// TIA Portal V16 export
// export: Created 2022-11-14T17:35:46.2709233Z, ExportSetting WithDefaults, DisplayName Totally Integrated Automation Portal, DisplayVersion V16, DisplayName TIA Portal Version Control Interface, DisplayVersion V16, DisplayName TIA Portal Openness, DisplayVersion V16, DisplayName STEP 7 Professional, DisplayVersion V16, DisplayName STEP 7 Safety, DisplayVersion V16, DisplayName WinCC Advanced, DisplayVersion V16
DATA_BLOCK "DB234_Program16"   // DB234
{ S7_Optimized_Access := 'FALSE' }
AUTHOR : Robopac
VERSION : 0.0
// stored: AutoNumber false, IsOnlyStoredInLoadMemory false, IsWriteProtectedInAS false
   VAR RETAIN
      Program16 { S7_SetPoint := 'True'} : "DatiProgramma";
   END_VAR
BEGIN
   Program16.Wrapping := FALSE;
   Program16.TopLenght := 0;
   Program16.TopRelease := 0;
   Program16.TopDown := 0;
   Program16.Top := 0;
   Program16.PressurePTime := 0;
   Program16.LifterTime := 0;
   Program16.RevOverContrast := 0;
   Program16.RopeEndCycle := 16#00;
   Program16.Spare4 := 16#00;
   Program16.RopeTime := 0;
   Program16.RevOverClamp := 0;
   Program16.FilmForceFinalRev := 0;
   Program16.FilmPrestretchFinalRev := 0;
   Program16.ArmSpeed := 0;
   Program16.CarriageDown4Top := 0;
   Program16.TopDownTime := 0;
   Program16.LapsUnderTop := 0;
   Program16.Spare6 := 0;
   Program16.Spare7 := 0;
   Program16.Spare8 := 0;
   Program16.Spare9 := 0;
   Program16.Spare10 := 0;
   Program16.Spare11 := 0;
   Program16.Spare12 := 0;
   Program16.Overlap0_1 := 0;
   Program16.Height1 := 0;
   Program16.Landmark1 := FALSE;
   Program16.Lifter1 := FALSE;
   Program16.SpareBit1H1 := FALSE;
   Program16.Airblower1 := FALSE;
   Program16.NextStep1 := FALSE;
   Program16.PressureP1 := FALSE;
   Program16.SpareByte2H1 := 16#00;
   Program16.Revolution1 := 0;
   Program16.RopeUnit1_1 := 16#00;
   Program16.RopeUnit1_2 := 16#00;
   Program16.FilmForce1 := 0;
   Program16.FilmPrestretch1 := 0;
   Program16.Spare3H1 := 0;
   Program16.Spare49 := 0;
   Program16.Spare50 := 0;
   Program16.Spare51 := 0;
   Program16.Spare52 := 0;
   Program16.Spare53 := 0;
   Program16.Overlap1_2 := 0;
   Program16.Height2 := 0;
   Program16.Landmark2 := FALSE;
   Program16.Lifter2 := FALSE;
   Program16.SpareBit1H2 := FALSE;
   Program16.Airblower2 := FALSE;
   Program16.NextStep2 := FALSE;
   Program16.PressureP2 := FALSE;
   Program16.SpareByte2H2 := 16#00;
   Program16.Revolution2 := 0;
   Program16.RopeUnit2_1 := 16#00;
   Program16.RopeUnit2_2 := 16#00;
   Program16.FilmForce2 := 0;
   Program16.FilmPrestretch2 := 0;
   Program16.Spare3H2 := 0;
   Program16.Spare54 := 0;
   Program16.Spare55 := 0;
   Program16.Spare56 := 0;
   Program16.Spare57 := 0;
   Program16.Spare58 := 0;
   Program16.Overlap2_3 := 0;
   Program16.Height3 := 0;
   Program16.Landmark3 := FALSE;
   Program16.Lifter3 := FALSE;
   Program16.SpareBit1H3 := FALSE;
   Program16.Airblower3 := FALSE;
   Program16.NextStep3 := FALSE;
   Program16.PressureP3 := FALSE;
   Program16.SpareByte2H3 := 16#00;
   Program16.Revolution3 := 0;
   Program16.RopeUnit3_1 := 16#00;
   Program16.RopeUnit3_2 := 16#00;
   Program16.FilmForce3 := 0;
   Program16.FilmPrestretch3 := 0;
   Program16.Spare3H3 := 0;
   Program16.Spare59 := 0;
   Program16.Spare60 := 0;
   Program16.Spare61 := 0;
   Program16.Spare62 := 0;
   Program16.Spare63 := 0;
   Program16.Overlap3_4 := 0;
   Program16.Height4 := 0;
   Program16.Landmark4 := FALSE;
   Program16.Lifter4 := FALSE;
   Program16.SpareBit1H4 := FALSE;
   Program16.Airblower4 := FALSE;
   Program16.NextStep4 := FALSE;
   Program16.PressureP4 := FALSE;
   Program16.SpareByte2H4 := 16#00;
   Program16.Revolution4 := 0;
   Program16.RopeUnit4_1 := 16#00;
   Program16.RopeUnit4_2 := 16#00;
   Program16.FilmForce4 := 0;
   Program16.FilmPrestretch4 := 0;
   Program16.Spare3H4 := 0;
   Program16.Spare64 := 0;
   Program16.Spare65 := 0;
   Program16.Spare66 := 0;
   Program16.Spare67 := 0;
   Program16.Spare68 := 0;
   Program16.Overlap4_5 := 0;
   Program16.Height5 := 0;
   Program16.Landmark5 := FALSE;
   Program16.Lifter5 := FALSE;
   Program16.SpareBit1H5 := FALSE;
   Program16.Airblower5 := FALSE;
   Program16.NextStep5 := FALSE;
   Program16.PressureP5 := FALSE;
   Program16.SpareByte2H5 := 16#00;
   Program16.Revolution5 := 0;
   Program16.RopeUnit5_1 := 16#00;
   Program16.RopeUnit5_2 := 16#00;
   Program16.FilmForce5 := 0;
   Program16.FilmPrestretch5 := 0;
   Program16.Spare3H5 := 0;
   Program16.Spare69 := 0;
   Program16.Spare70 := 0;
   Program16.Spare71 := 0;
   Program16.Spare72 := 0;
   Program16.Spare73 := 0;
   Program16.Overlap5_6 := 0;
   Program16.Height6 := 0;
   Program16.Landmark6 := FALSE;
   Program16.Lifter6 := FALSE;
   Program16.SpareBit1H6 := FALSE;
   Program16.Airblower6 := FALSE;
   Program16.NextStep6 := FALSE;
   Program16.PressureP6 := FALSE;
   Program16.SpareByte2H6 := 16#00;
   Program16.Revolution6 := 0;
   Program16.RopeUnit6_1 := 16#00;
   Program16.RopeUnit6_2 := 16#00;
   Program16.FilmForce6 := 0;
   Program16.FilmPrestretch6 := 0;
   Program16.Spare3H6 := 0;
   Program16.Spare74 := 0;
   Program16.Spare75 := 0;
   Program16.Spare76 := 0;
   Program16.Spare77 := 0;
   Program16.Spare78 := 0;
   Program16.Overlap6_7 := 0;
   Program16.Height7 := 0;
   Program16.Landmark7 := FALSE;
   Program16.Lifter7 := FALSE;
   Program16.SpareBit1H7 := FALSE;
   Program16.Airblower7 := FALSE;
   Program16.NextStep7 := FALSE;
   Program16.PressureP7 := FALSE;
   Program16.SpareByte2H7 := 16#00;
   Program16.Revolution7 := 0;
   Program16.RopeUnit7_1 := 16#00;
   Program16.RopeUnit7_2 := 16#00;
   Program16.FilmForce7 := 0;
   Program16.FilmPrestretch7 := 0;
   Program16.Spare3H7 := 0;
   Program16.Spare79 := 0;
   Program16.Spare80 := 0;
   Program16.Spare81 := 0;
   Program16.Spare82 := 0;
   Program16.Spare83 := 0;
   Program16.Overlap7_8 := 0;
   Program16.Height8 := 0;
   Program16.Landmark8 := FALSE;
   Program16.Lifter8 := FALSE;
   Program16.SpareBit1H8 := FALSE;
   Program16.Airblower8 := FALSE;
   Program16.NextStep8 := FALSE;
   Program16.PressureP8 := FALSE;
   Program16.SpareByte2H8 := 16#00;
   Program16.Revolution8 := 0;
   Program16.RopeUnit8_1 := 16#00;
   Program16.RopeUnit8_2 := 16#00;
   Program16.FilmForce8 := 0;
   Program16.FilmPrestretch8 := 0;
   Program16.Spare3H8 := 0;
   Program16.Spare84 := 0;
   Program16.Spare85 := 0;
   Program16.Spare86 := 0;
   Program16.Spare87 := 0;
   Program16.Spare88 := 0;
   Program16.Overlap8_9 := 0;
   Program16.Height9 := 0;
   Program16.Landmark9 := FALSE;
   Program16.Lifter9 := FALSE;
   Program16.SpareBit1H9 := FALSE;
   Program16.Airblower9 := FALSE;
   Program16.NextStep9 := FALSE;
   Program16.PressureP9 := FALSE;
   Program16.SpareByte2H9 := 16#00;
   Program16.Revolution9 := 0;
   Program16.RopeUnit9_1 := 16#00;
   Program16.RopeUnit9_2 := 16#00;
   Program16.FilmForce9 := 0;
   Program16.FilmPrestretch9 := 0;
   Program16.Spare3H9 := 0;
   Program16.Spare89 := 0;
   Program16.Spare90 := 0;
   Program16.Spare91 := 0;
   Program16.Spare92 := 0;
   Program16.Spare93 := 0;
   Program16.Overlap9_10 := 0;
   Program16.Height10 := 0;
   Program16.Landmark10 := FALSE;
   Program16.Lifter10 := FALSE;
   Program16.SpareBit1H10 := FALSE;
   Program16.Airblower10 := FALSE;
   Program16.NextStep10 := FALSE;
   Program16.PressureP10 := FALSE;
   Program16.SpareByte2H10 := 16#00;
   Program16.Revolution10 := 0;
   Program16.RopeUnit10_1 := 16#00;
   Program16.RopeUnit10_2 := 16#00;
   Program16.FilmForce10 := 0;
   Program16.FilmPrestretch10 := 0;
   Program16.Spare3H10 := 0;
   Program16.Spare94 := 0;
   Program16.Spare95 := 0;
   Program16.Spare96 := 0;
   Program16.Spare97 := 0;
   Program16.Spare98 := 0;
   Program16.Overlap10_11 := 0;
   Program16.Height11 := 0;
   Program16.Landmark11 := FALSE;
   Program16.Lifter11 := FALSE;
   Program16.SpareBit1H11 := FALSE;
   Program16.Airblower11 := FALSE;
   Program16.NextStep11 := FALSE;
   Program16.PressureP11 := FALSE;
   Program16.SpareByte2H11 := 16#00;
   Program16.Revolution11 := 0;
   Program16.RopeUnit11_1 := 16#00;
   Program16.RopeUnit11_2 := 16#00;
   Program16.FilmForce11 := 0;
   Program16.FilmPrestretch11 := 0;
   Program16.Spare3H11 := 0;
   Program16.Spare99 := 0;
   Program16.Spare100 := 0;
   Program16.Spare101 := 0;
   Program16.Spare102 := 0;
   Program16.Spare103 := 0;
   Program16.Overlap11_12 := 0;
   Program16.Height12 := 0;
   Program16.Landmark12 := FALSE;
   Program16.Lifter12 := FALSE;
   Program16.SpareBit1H12 := FALSE;
   Program16.Airblower12 := FALSE;
   Program16.NextStep12 := FALSE;
   Program16.PressureP12 := FALSE;
   Program16.SpareByte2H12 := 16#00;
   Program16.Revolution12 := 0;
   Program16.RopeUnit12_1 := 16#00;
   Program16.RopeUnit12_2 := 16#00;
   Program16.FilmForce12 := 0;
   Program16.FilmPrestretch12 := 0;
   Program16.Spare3H12 := 0;
   Program16.Spare104 := 0;
   Program16.Spare105 := 0;
   Program16.Spare106 := 0;
   Program16.Spare107 := 0;
   Program16.Spare108 := 0;
END_DATA_BLOCK
